// TIA Portal V17 export
// export: Created 2023-08-28T22:41:32.6164324Z, ExportSetting WithDefaults, DisplayName Totally Integrated Automation Portal, DisplayVersion V17 Update 5, DisplayName TIA Portal Openness, DisplayVersion V17 Update 5, DisplayName TIA Portal Teamcenter Gateway, DisplayVersion V17 Update 5, DisplayName TIA Portal Version Control Interface, DisplayVersion V17, DisplayName Simotion SCOUT TIA, DisplayVersion 5.4.3.0, DisplayName TIA Portal Test Suite Advanced, DisplayVersion V17 Update 1, DisplayName SIMOCODE ES, DisplayVersion V17 Update 5, DisplayName SINAMICS Startdrive Advanced, DisplayVersion V17 SP1, DisplayName SINAMICS Startdrive G130, G150, S120, S150, SINAMICS MV, S210, DisplayVersion V17 SP1, DisplayName SINAMICS Startdrive G110M, G120, G120C, G120D, G120P, G115D, DisplayVersion V17 SP1, DisplayName SIRIUS Safety ES, DisplayVersion V17 Update 5, DisplayName STEP 7 Professional, DisplayVersion V17 Update 5, DisplayName STEP 7 CFC, DisplayVersion V17 Update 1, DisplayName STEP 7 Safety, DisplayVersion V17, DisplayName WinCC Advanced, DisplayVersion V17 Update 5, DisplayName SIMATIC Visualization Architect, DisplayVersion V17 Update 5
DATA_BLOCK "n0013-uf317-xn10_SN50_1"   // DB27, F_DB
VERSION : 0.1
// stored: AutoNumber true, DBAccessibleFromOPCUA true, DBAccessibleFromWebserver true, InstanceOfName 00_Push-Button_Input, InstanceOfType FB
"00_Push-Button_Input"
   // VAR_INPUT
   //    IN_1 : Bool;
   //    IN_2 : Bool;
   //    IN_3 : Bool;
   //    IN_4 : Bool;
   //    ON_Tristate : Bool;
   //    ON_Lamp : Bool;
   //    Reset : Bool;
   //    REAC_DELAY { ExternalWritable := 'False'} : Time;
   //    Bypass_ET200 : Bool;
   // END_VAR
   // VAR_OUTPUT
   //    OUT_1 : Bool;
   //    OUT_2 : Bool;
   //    OUT_3 : Bool;
   //    OUT_4 : Bool;
   //    Diag_1 : Bool;
   //    Diag_2 : Bool;
   //    Diag_3 : Bool;
   //    Diag_4 : Bool;
   //    Lamp_1 : Bool;
   //    Lamp_2 : Bool;
   //    Lamp_3 : Bool;
   //    Lamp_4 : Bool;
   // END_VAR
   // VAR
   //    ESTOP_1 { S7_SetPoint := 'True'} : ESTOP1;
   //    ESTOP_2 { S7_SetPoint := 'True'} : ESTOP1;
   //    ESTOP_3 { S7_SetPoint := 'True'} : ESTOP1;
   //    ESTOP_4 { S7_SetPoint := 'True'} : ESTOP1;
   //    TON_1 { ExternalWritable := 'False'} : TON;
   //    TON_2 { ExternalWritable := 'False'} : TON;
   //    TON_3 { ExternalWritable := 'False'} : TON;
   //    TON_4 { ExternalWritable := 'False'} : TON;
   // END_VAR
BEGIN
END_DATA_BLOCK
